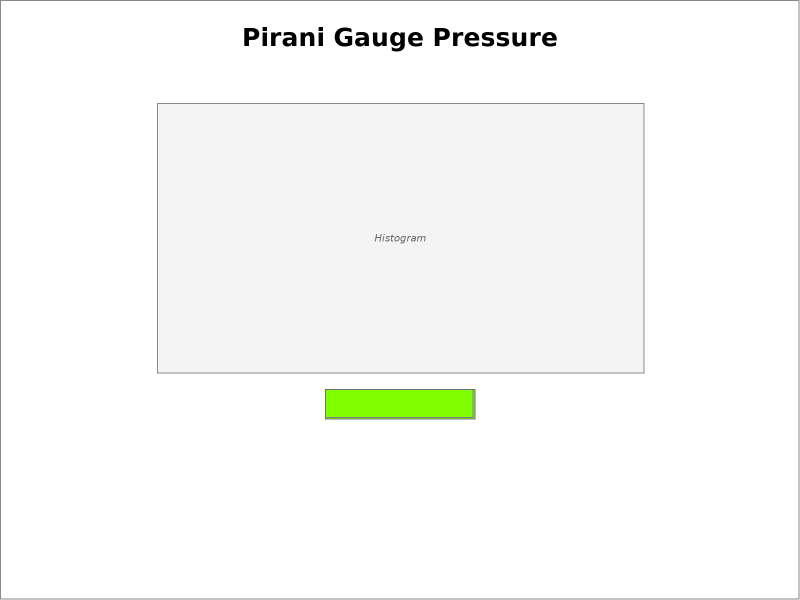
VISUALIZATION Visualization  // 800x600
    Label (160,5 480x64), "Pirani Gauge Pressure"
    Histogram (157,103 487x270), scale format: %.1f, scale 0..100
    Button (325,389 150x30)
END_VISUALIZATION

(* stored: Version 1.1.0.1
   Visu Visualization: Id {7e560e81-f1ab-4d55-9410-0415b15fbbc8} *)
